// TIA Portal V19 export
VAR_GLOBAL   // PLC tag table "LAcycCom_Common"
END_VAR
VAR_GLOBAL CONSTANT   // user constants
   LACYCCOM_BUFFER_ELEMENTS_UPPER_LIM : Int := 59;   // Upper limit of request buffer array
END_VAR
